TYPE ST_SequenceOut :
STRUCT
END_STRUCT
END_TYPE

(* stored: Version 1.1.0.1
   DUT ST_SequenceOut: Id {bef8f698-fe05-0dc0-22ca-45ad7ad730f3} *)
